FUNCTION_BLOCK InputChannelAdptd (* Composite Function Block Type *)
  (* Standard: 61499-2 *)
  (* Version 0.0, 09/10/2018, Atmojo, nxtControl GmbH, template *)
  PACKAGE Main;
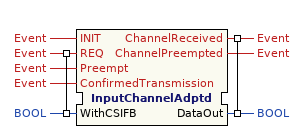
  EVENT_INPUT
    INIT;
    REQ WITH WithCSIFB; (* Normal Execution Request *)
    Preempt; (* Initialization Request *)
    ConfirmedTransmission;
  END_EVENT
  EVENT_OUTPUT
    ChannelReceived WITH DataOut; (* Initialization Confirm *)
    ChannelPreempted; (* Execution Confirmation *)
  END_EVENT
  VAR_INPUT
    WithCSIFB : BOOL;
  END_VAR
  VAR_OUTPUT
    DataOut : BOOL;
  END_VAR
END_FUNCTION_BLOCK
